TYPE STRUCT_EVENT :
STRUCT
	_ID:				UINT;
	_VAL1:			STRING;
	_VAL2:			STRING;
	_VAL3:			STRING;
	_HORODAT:		DT;
	_MS:			UINT;
	_TYPE:			BOOL;	(*True = apparition, False=disparition*)
END_STRUCT
END_TYPE

(* stored: Version 1.1.0.1, ProductVersion 3.1.4024.10
   DUT STRUCT_EVENT: Id {176b59a0-234a-4f8c-9576-eb9a7e6d9507} *)
